//{attribute 'qualified_only'}
VAR_GLOBAL //data arrays to be passed into material holder FBs - do not access directly
	skidHmiA22Left : ARRAY[1...Cardboard.size-1] OF MaterialSlot;
	skidHmiA22Right : ARRAY[1...Cardboard.size-1] OF MaterialSlot;
	
	magazineHmiA22Left : ARRAY[1..CornerGuard.size-1] OF MaterialSlot;
	magazineHmiA22Right : ARRAY[1..CornerGuard.size-1] OF MaterialSlot;
END_VAR

(* stored: Version 1.1.0.1, ProductVersion 3.1.4024.11
   GVL ContainerArrays: Id {a41ac828-3b90-4453-b6ae-c19c2ca38393} *)
